//============================================================================
// Author: Dereje Hailemariam
// Datum: 27.08.2026
// Version: 2.2 — Vision at 2-axis P&P (pre-assembly) → RFID write later
//
// Hardware:
//   Vision cameras at Zone 3B 2-axis Pick & Place (lid + base BEFORE assembly)
//   RFID Reader 2 at pallet / 4b write station
//
// Sequence:
//   Vision latch at P&P → assembly → 4b_Done → Write_Req → tag pallet
//============================================================================

ORGANIZATION_BLOCK "OB1_Main"
{ S7_Optimized_Access := 'TRUE' }
VERSION : 2.2

BEGIN
    //------------------------------------------------------------------
    // 1) Vision — sense at 2-axis P&P; write only when Allow_Write
    //------------------------------------------------------------------
    "FB_VisionReader_Plastic"(
        Enable                      := TRUE,
        Vision_Lid_Value            := "2b_Vision Sensor Lid (Value)",
        Vision_Base_Value           := "2b_Vision Sensor Base(Value)",

        // Pallet ready for RFID (after assembly / palletizer Done)
        Allow_Write                 := "4b_Done(1)",

        RFID_Bereit                 := "2b_HMI_RFID_Bereit",
        RFID_Busy                   := "2b_HMI_RFID_Busy",
        RFID_Done                   := "2b_HMI_RFID_Done",
        Reset                       := "2b_HMI_RFID_Reset",

        Both_Ready                  => "2b_VisionData_Both_Ready",
        Color_Code                  => "2b_VisionData_Color_Code",

        Materialart                 => "2b_VisionData_Materialart",
        ProductTyp                  => "2b_VisionData_ProductType",
        Artikelnummer               => "2b_VisionData_Artikelnumber",
        RFID_Code                   => "2b_VisionData_RFID_CODE",

        Write_Req                   => "2b_HMI_RFID_Write",
        Combo_Done                  => "2b_VisionData_Combo_Done",
        Busy                        => "Vision_Busy",
        Waiting_For_Write           => "2b_VisionData_Waiting_For_Write",
        Error                       => "Vision_Error",
        State                       => "2b_VisionData_State"
    );

    //------------------------------------------------------------------
    // 2) RFID WRITE — Reader 2 (Vision Write_Req only)
    //------------------------------------------------------------------
    "RFID_Read_Write_DB_1"(
        Execute                     := FALSE,
        HMI_Read                    := FALSE,
        HMI_Write                   := "2b_HMI_RFID_Write",
        HMI_Check                   := FALSE,
        HMI_Clear                   := FALSE,
        HMI_Reset                   := "2b_HMI_RFID_Reset",
        RFID_Lesen                  := FALSE,

        Op_Mode                     := 10,

        Command_ID                  := "4b_RFID Reader 2 Command ID",
        Status                      := "4b_RFID Reader 2 Status",
        Read_Data                   := "4b_RFID Reader 2 Read Data",

        Memory_Index                := 0,
        Write_Data                  := 0,

        RFID_Code_In                := "2b_VisionData_RFID_CODE",
        Artikelnummer_In            := "2b_VisionData_Artikelnumber",
        Materialart_In              := "2b_VisionData_Materialart",
        ProductTyp_In               := "2b_VisionData_ProductType",

        Timeout                     := T#15S,
        Tag_Wait_Time               := T#3M,
        Execute_Hold                := T#100MS,

        Execute_Command             => "4b_RFID Reader 2 Execute Command",
        Command                     => "4b_RFID Reader 2 Command",
        Memory_Index_Out            => "4b_RFID Reader 2 Memory Index",
        Write_Data_Out              => "4b_RFID Reader 2 Write Data",

        Busy                        => "2b_HMI_RFID_Busy",
        Done                        => "2b_HMI_RFID_Done",
        Error                       => "RFID_Error",
        Status_Code                 => "RFID_Status_Code",

        RFID_Bereit                 => "2b_HMI_RFID_Bereit",
        RFID_Gueltig                => "RFID_Gueltig",
        RFID_Fehler                 => "RFID_Fehler",

        RFID_Code_Out               => "RFID_Code_Out",
        Artikelnummer_Out           => "RFID_Artikelnummer_Out",
        Materialart_Out             => "RFID_Materialart_Out",
        ProductTyp_Out              => "RFID_ProductTyp_Out",

        Pallet_Tagged               => "2b_HMI_RFID_Pallet_Tagged"
    );

END_ORGANIZATION_BLOCK
